FUNCTION_BLOCK HTTP_POST_JSON
  {SET_ATTRIBUTE(OpcUa, POINT.ENDPOINT)}
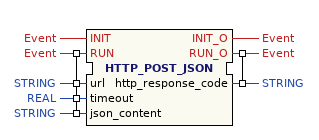
  EVENT_INPUT
    INIT;
    RUN WITH url, timeout, json_content; {SET_ATTRIBUTE(OpcUa, Method)}
  END_EVENT
  EVENT_OUTPUT
    INIT_O;
    RUN_O WITH http_response_code;
  END_EVENT
  VAR_INPUT
    url : STRING; {SET_ATTRIBUTE(OpcUa, Variable.RUN)}
    timeout : REAL; {SET_ATTRIBUTE(OpcUa, Variable.RUN)}
    json_content : STRING; {SET_ATTRIBUTE(OpcUa, Variable.RUN)}
  END_VAR
  VAR_OUTPUT
    http_response_code : STRING; {SET_ATTRIBUTE(OpcUa, Variable.RUN)}
  END_VAR
END_FUNCTION_BLOCK
